(* CoDeSys 2.3 project: LAB3_HMI (1).pro *)
(* Libraries: IECSFC_S90_V41.lib 7.6.00 16:18:20, IEC_S90_V41.LIB 11.4.02 10:16:10 *)

(* Global variable list: Auslastung *)
VAR_GLOBAL
	Auslastung AT %MW1259.0 :INT;
	TaskID_verfehlte_Zyklen AT %MW1259.1:INT;
	Verfehlte_ms AT %MW1259.2:INT;
	VerfehlteZyklen AT %MW1259.3 : INT;
	SuspendierteTasks AT %MW1259.4 : INT;
END_VAR

(* Global variable list: Fehlermerker *)
VAR_GLOBAL
	M255_00 AT %MX255.0 : BOOL;
	M255_01 AT %MX255.1 : BOOL;
	M255_02 AT %MX255.2 : BOOL;
	M255_03 AT %MX255.3 : BOOL;
	M255_04 AT %MX255.4 : BOOL;
	M255_05 AT %MX255.5 : BOOL;
	M255_06 AT %MX255.6 : BOOL;
	M255_07 AT %MX255.7 : BOOL;
	M255_08 AT %MX255.8 : BOOL;
	M255_09 AT %MX255.9 : BOOL;
	M255_10 AT %MX255.10 : BOOL;
	M255_11 AT %MX255.11 : BOOL;
	M255_12 AT %MX255.12 : BOOL;
	M255_13 AT %MX255.13 : BOOL;
	M255_14 AT %MX255.14 : BOOL;
	M255_15 AT %MX255.15 : BOOL;
	MW254_00 AT %MW1254.0 : INT;
	MW254_01 AT %MW1254.1 : INT;
	MW254_02 AT %MW1254.2 : INT;
	MW254_03 AT %MW1254.3 : INT;
	MW254_04 AT %MW1254.4 : INT;
	MW254_05 AT %MW1254.5 : INT;
	MW254_06 AT %MW1254.6 : INT;
	MW254_07 AT %MW1254.7 : INT;
	MW254_08 AT %MW1254.8 : INT;
	MW254_09 AT %MW1254.9 : INT;
	MW254_10 AT %MW1254.10 : INT;
	MW254_11 AT %MW1254.11 : INT;
	MW254_12 AT %MW1254.12 : INT;
	MW254_13 AT %MW1254.13 : INT;
	MW254_14 AT %MW1254.14 : INT;
	MW254_15 AT %MW1254.15 : INT;
	MW255_00 AT %MW1255.0 : INT;
	MW255_01 AT %MW1255.1 : INT;
	MW255_02 AT %MW1255.2 : INT;
	MW255_03 AT %MW1255.3 : INT;
	MW255_04 AT %MW1255.4 : INT;
	MW255_05 AT %MW1255.5 : INT;
	MW255_06 AT %MW1255.6 : INT;
	MW255_07 AT %MW1255.7 : INT;
	MW255_08 AT %MW1255.8 : INT;
	MW255_09 AT %MW1255.9 : INT;
	MW255_10 AT %MW1255.10 : INT;
	MW255_11 AT %MW1255.11 : INT;
	MW255_12 AT %MW1255.12 : INT;
	MW255_13 AT %MW1255.13 : INT;
	MW255_14 AT %MW1255.14 : INT;
	MW255_15 AT %MW1255.15 : INT;
END_VAR

(* Global variable list: Systemkonstanten *)
VAR_GLOBAL
(* Standard - Systemkonstanten *)
(* -1 Master / -2 Standalone / 0..61 Slave *)
	KW00_00 AT %MW3000.0 : INT := -2;
(* Pufferung Binärmerker %MX000.00-%MX511.15 *)
	KW00_01 AT %MW3000.1 : INT := 0 ;
(* Pufferung Wortmerker %MW1000.00-%MW1511.15 *)
	KW00_02 AT %MW3000.2 : INT := 0 ;
(* Pufferung Doppelwortmerker %MW2000.00-%MW2063.15 *)
	KW00_03 AT %MW3000.3 : INT := 0 ;
(* Pufferung Schrittkettenmerker %MW5000-%MW5255 *)
	KW00_04 AT %MW3000.4 : INT := 0 ;
	KW00_05 AT %MW3000.5 : INT := 0 ;
	KW00_06 AT %MW3000.6 : INT := 0 ;
(* SPS-Reaktion auf Fehler der Klasse 3 *)
	KW00_07 AT %MW3000.7 : INT := 0 ;
	KW00_08 AT %MW3000.8 : INT := 0 ;
	KW00_09 AT %MW3000.9 : INT := 0 ;
(* Größe des Sendebereichs der Slave-SPS *)
	KW00_10 AT %MW3000.10 : INT := 0 ;
(* Größe des Empfangsbereiches der Slave-SPS *)
	KW00_11 AT %MW3000.11 : INT := 0 ;
(* Automatischer Warmstart nach FK2-Fehler *)
	KW00_12 AT %MW3000.12 : INT := 0 ;
	KW00_13 AT %MW3000.13 : INT := 0 ;
	KW00_14 AT %MW3000.14 : INT := 0 ;
(* Oszillatoren auf %MX255.0-%MX255.6 deaktivieren *)
	KW00_15 AT %MW3000.15 : INT := 0 ;
(* Überwachung der Task mit Zykluszeit > 0 *)
	KW80_00 AT %MW3080.0 : INT := 0;
(* Überwachung der Task mit Zykluszeit = 0 *)
	KW80_01 AT %MW3080.1 : INT := 0;
(*Bit stellt Eingangsverzögerung fuer E62_00 bis E62_15 ein: 1=1ms, 0=7ms*)
	KW85_00 AT %MW3085.0 : INT := 0;
(*Bit stellt Eingangsverzögerung fuer E63_00 bis E63_15 ein: 1=1ms, 0=7ms*)
	KW85_01 AT %MW3085.1 : INT := 0;
(*Konfiguriert die Zaehlebetriebsart E62_00, E62_01 und A62_00 (siehe unten)*)
	KW85_02 AT %MW3085.2 : INT := 0;
	KW85_03 AT %MW3085.3 : INT := 0;
	KW85_04 AT %MW3085.4 : INT := 0;
	KW85_05 AT %MW3085.5 : INT := 0;
	KW85_06 AT %MW3085.6 : INT := 0;
	KW85_07 AT %MW3085.7 : INT := 0;
	KW85_08 AT %MW3085.8 : INT := 0;
	KW85_09 AT %MW3085.9 : INT := 0;
	KW85_10 AT %MW3085.10 : INT := 0;
	KW85_11 AT %MW3085.11 : INT := 0;
	KW85_12 AT %MW3085.12 : INT := 0;
	KW85_13 AT %MW3085.13 : INT := 0;
	KW85_14 AT %MW3085.14 : INT := 0;
	KW85_15 AT %MW3085.15 : INT := 0;
(*Konfiguriert Analogeingang EW06_00 (siehe unten)*)
	KW86_00 AT %MW3086.0 : INT := 0;
(*Konfiguriert Analogeingang EW06_01 (siehe unten)*)
	KW86_01 AT %MW3086.1 : INT := 0;
(*Konfiguriert Analogeingang EW06_02 (siehe unten)*)
	KW86_02 AT %MW3086.2 : INT := 0;
(*Konfiguriert Analogeingang EW06_03 (siehe unten)*)
	KW86_03 AT %MW3086.3 : INT := 0;
(*Konfiguriert Analogeingang EW06_04 (siehe unten)*)
	KW86_04 AT %MW3086.4 : INT := 0;
(*Konfiguriert Analogeingang EW06_05 (siehe unten)*)
	KW86_05 AT %MW3086.5 : INT := 0;
(*Konfiguriert Analogeingang EW06_06 (siehe unten)*)
	KW86_06 AT %MW3086.6 : INT := 0;
(*Konfiguriert Analogeingang EW06_07 (siehe unten)*)
	KW86_07 AT %MW3086.7 : INT := 0;
	KW86_08 AT %MW3086.8 : INT := 0;
	KW86_09 AT %MW3086.9 : INT := 0;
	KW86_10 AT %MW3086.10 : INT := 0;
	KW86_11 AT %MW3086.11 : INT := 0;
	KW86_12 AT %MW3086.12 : INT := 0;
	KW86_13 AT %MW3086.13 : INT := 0;
	KW86_14 AT %MW3086.14 : INT := 0;
	KW86_15 AT %MW3086.15 : INT := 0;
(*Konfiguriert Analogausgang AW06_00 (siehe unten)*)
	KW88_00 AT %MW3088.0 : INT := 0;
(*Konfiguriert Analogausgang AW06_01 (siehe unten)*)
	KW88_01 AT %MW3088.1 : INT := 0;
(*Konfiguriert Analogausgang AW06_02 (siehe unten)*)
	KW88_02 AT %MW3088.2 : INT := 0;
(*Konfiguriert Analogausgang AW06_03 (siehe unten)*)
	KW88_03 AT %MW3088.3 : INT := 0;

(* Zykluszeit in [ms]
 ACHTUNG: WIRD NICHT MEHR UNTERSTUETZT; STATT DESSEN TASKKONFIGURATION *)
	ZyklusZeit AT %MD4000.0 : DWORD;
END_VAR

(*Konfiguration der Analogeingaenge EW06_00 bis EW06_07 ueber KW86_00 bis KW86_07*)
(*Low-Byte der KW*)
(*0x00		Analogeingang 0...10V (Standardeinstellung)*)
(*0x01		nicht benutzt*)
(*0x02		Digitaler Eingang mit 7ms Eingangsverzögerung*)
(*0x03		Analogeingang 0..20mA*)
(*0x04		Analogeingang 4..20mA*)
(*0x05		Analogeingang -10V..+10V*)
(*0x06		Analogeingang 0V..5V*)
(*0x07		Analogeingang -5V..+5V*)
(*0x08		Analogeingang Pt100 in 2-Draht-Anschluß -50°C..+400°C*)
(*0x09		Analogeingang Pt100 in 3-Draht-Anschluß -50°C..+400°C*)
(*0x0A		Analogeingang 0V..10V Differenzeingang*)
(*0x0B		Analogeingang -10V..+10V Differenzeingang*)
(*0x0C		Analogeingang 0V..5V Differenzeingang*)
(*0x0D		Analogeingang -5V..+5V Differenzeingang*)
(*0x0E		Analogeingang Pt100 in 2-Draht-Anschluß -50°C..+70°C*)
(*0x0F		Analogeingang Pt100 in 3-Draht-Anschluß -50°C..+70°C*)
(*High-Byte der KW*)
(*0x00		Plausibilitaetsueberwachung und Drahtbruch- und Kurzschlußueberwachung (Standard)*)
(*0x01		Drahtbruch- und Kurzschlußueberwachung*)
(*0x02		Plausibilitaetsueberwachung*)
(*0x03		Keine Ueberwachung*)

(*Konfiguration der Analogausgaenge AW06_00 bis AW06_03 ueber KW88_00 bis KW88_03*)
(*Low-Byte der KW*)
(*0x00		Analogausgang -10V..+10V (Standardeinstellung)*)
(*0x01		nicht benutzt*)
(*0x02		Analogausgang 0..20mA*)
(*0x03		Analogausgang 4..20mA*)

(*Konfiguration der Zaehlerbetriebsart E62_00, E62_01und A62_00 ueber KW85_02*)
(*Low-Byte der KW*)
(*0x00		Kein Zaehler (Standardeinstellung)*)
(*0x01		Mode 1,	Ein Vorwaertszaehler*)
(*0x02		Mode 2,	Ein Vorwaertszaehler mit Freigabeeingang*)
(*0x03		Mode 3,	Zwei Vorwaerts-/Rueckwaertszaehler*)
(*0x04		Mode 4,	Zwei Vorwaerts-/Rueckwaertszaehler;*)
(*						der zweite Zaehler zaehlt die Impulse der fallenden Flanke*)
(*0x05		Mode 5,	Ein Vorwaerts-/Rueckwaertszaehler mit dynamischem Setzeingang,*)
(*						Setzen auf steigender Flanke*)
(*0x06		Mode 6,	Ein Vorwaerts-/Rueckwaertszaehler mit dynamischem Setzeingang,*)
(*						Setzen auf fallender Flanke*)
(*0x07		Mode 7,	Ein Vorwaerts-/Rueckwaertszaehler mit Richtungsdiskriminator*)

(* POU PLC_PRG, SFC *)
PROGRAM PLC_PRG
VAR
	INICIO AT %IX62.0: BOOL;
	SA1: BOOL;
	SB1: BOOL;
	SC1: BOOL;
	SB2: BOOL;
	CA AT %QX62.0: BOOL;
	CB AT %QX62.1: BOOL;
	CC AT %QX62.2: BOOL;

	RETARDO: BOOL;

	XA: REAL := 0;
	XA2: REAL := 0;
       YA2: REAL := 0;
	XB: REAL := 0;
      YB: REAL := 0;
	XC: REAL := 0;
      YC: REAL := 0;
      VELA: REAL := 3;
	R1: BOOL;
	R2:BOOL;
END_VAR
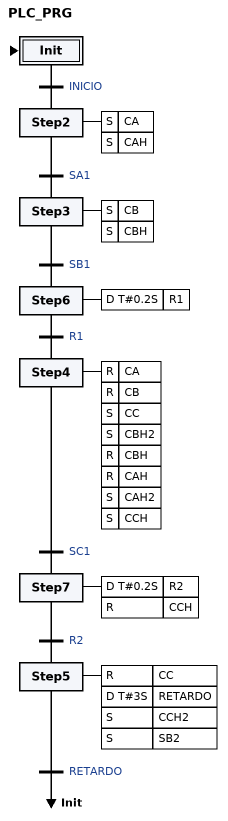
INITIAL_STEP Init:
END_STEP
TRANSITION FROM Init TO Step2 := INICIO;
END_TRANSITION
STEP Step2:
	CA(S);
	CAH(S);
END_STEP
TRANSITION FROM Step2 TO Step3 := SA1;
END_TRANSITION
STEP Step3:
	CB(S);
	CBH(S);
END_STEP
TRANSITION FROM Step3 TO Step6 := SB1;
END_TRANSITION
STEP Step6:
	R1(D, T#0.2S);
END_STEP
TRANSITION FROM Step6 TO Step4 := R1;
END_TRANSITION
STEP Step4:
	CA(R);
	CB(R);
	CC(S);
	CBH2(S);
	CBH(R);
	CAH(R);
	CAH2(S);
	CCH(S);
END_STEP
TRANSITION FROM Step4 TO Step7 := SC1;
END_TRANSITION
STEP Step7:
	R2(D, T#0.2S);
	CCH(R);
END_STEP
TRANSITION FROM Step7 TO Step5 := R2;
END_TRANSITION
STEP Step5:
	CC(R);
	RETARDO(D, T#3S);
	CCH2(S);
	SB2(S);
END_STEP
TRANSITION FROM Step5 TO Init := RETARDO;
END_TRANSITION
END_PROGRAM
ACTION CAH:
IF XA<= 150 THEN
XA := XA + VELA;
XA2:= XA2+ VELA;
END_IF

IF XA >= 150 THEN
SA1 := TRUE;
ELSE
SA1 := FALSE;
END_IF
END_ACTION
ACTION CAH2:
IF XA>=0 THEN
XA := XA-VELA;
END_IF

IF XA <= 150 THEN
SA1 := FALSE;
ELSE
SA1 := TRUE;
END_IF
END_ACTION
ACTION CBH:
IF YB<=150 THEN
YB:= YB+VELA;
END_IF
IF XB<= 150 THEN
XB:= XB + VELA;
END_IF

IF XB>=150 THEN
SB1:= TRUE;
ELSE
SB1:= FALSE;
END_IF
END_ACTION
ACTION CBH2:
IF YB>=0 THEN
YB:= YB-VELA;
END_IF
IF XB>=0 THEN
XB:= XB-VELA;
END_IF
IF XB<=150 THEN
SB1:= FALSE;
ELSE
SB1:= TRUE;
END_IF
END_ACTION
ACTION CCH:
SB2:=TRUE;
IF YC<=700 THEN
YC:= YC+VELA;
END_IF
IF XC<= 150 THEN
XC:= XC + VELA;
END_IF

IF XC>=150 THEN
SC1:= TRUE;
ELSE
SC1:= FALSE;
END_IF
END_ACTION
ACTION CCH2:
SB2:=TRUE;
IF YC>=0 THEN
YC:= YC-VELA;
END_IF
IF XC>=0 THEN
XC:= XC - VELA;
END_IF
IF YA2<=150 THEN
YA2:= YA2+ 9;
END_IF

IF XC>=150 THEN
SC1:= TRUE;
ELSE
SC1:= FALSE;
END_IF
END_ACTION
